{attribute 'qualified_only'}
{attribute 'strict'}
TYPE JoystickCalibState :
(
	CalibMinMax := 0,
	CalibDeadband := 1,
	CalibOver := 2,
	CalibStart := 3
);
END_TYPE

(* stored: Version 1.1.0.1, ProductVersion 3.1.4022.18
   DUT JoystickCalibState: Id {6ac9e214-d654-494f-bb52-97e0f6cac6b9} *)
